(* CoDeSys 2.3.9.41 project: A1.pro *)
(* Libraries: STANDARD.LIB*16.9.21 10:31:38, IECSFC.LIB*16.9.21 10:31:38, SYSLIBTIME.LIB*16.9.21 10:31:38, SYSTASKINFO.LIB*16.9.21 10:31:38, ANALYZATION.LIB*16.9.21 10:31:38, SYSLIBCALLBACK.LIB*16.9.21 10:31:38, Util.lib*16.9.21 10:31:38 *)

(* PLC configuration (modules and I/O channels)
DI_1 AT %IX0.0 [BitInput] Discrete input 1 {ChannellName = Enter name}
DI_2 AT %IX0.1 [BitInput] Discrete input 2 {ChannellName = Enter name}
AT %IB1.0 [ByteInput] 8 discrete inputs {ChannellName = Enter name}
AT %IB1.1 [ByteInput] 8 discrete inputs {ChannellName = Enter name}
DO_1 AT %QX2.0 [BitOutput] Fast discrete output 1 {ChannellName = Enter name}
DO_2 AT %QX2.1 [BitOutput] Fast discrete output 2 {ChannellName = Enter name}
DO_3 AT %QX2.2 [BitOutput] Fast discrete output 3 {ChannellName = Enter name}
DO_4 AT %QX2.3 [BitOutput] Fast discrete output 4 {ChannellName = Enter name}
AT %QB3.0 [ByteOutput] 8 discrete outputs {ChannellName = Enter name}
AT %QB3.1 [ByteOutput] 8 discrete outputs {ChannellName = Enter name}
Special input [ID103] node 4, in %IB4 out %QB4 {ChannellName = Special input}
  AT %IX4.0 [BitInput] Special input {ChannellName = Enter name}
Special output [ID104] node 5, in %IB5 out %QB5 {ChannellName = Special output}
  AT %QX5.0 [BitOutput] Special output {ChannellName = Enter name}
AT %QD6.0 [DWordOutput] Last address {ChannellName = Enter name}
AT %QW6.1 [WordOutput] Last error {ChannellName = Enter name}
RS-485-1 [COM1_USART] node 0, in %IB6.0 out %QB6.0 {ChannellName = RS-485-1; CommunicationSpeed = 115200; Parity = NO PARITY CHECK; BitLength = 8 bits; StopLength = One stop bit; InterfaceType = RS485; FrameOriented = RTU; Timeout = 0; Visibility = No}
AT %QB6.1.0 [ComChannel] Command (0xff - Start) {ChannellName = Enter name}
AlarmA2 AT %QW6.1.0.0 [WordOutput] {ChannellName = Enter name}
qNeedPressure1 AT %QW6.1.1.0 [WordOutput] {ChannellName = Enter name}
qNeedPressure2 AT %QW6.1.2.0 [WordOutput] {ChannellName = Enter name}
qNeedPressure3 AT %QW6.1.3.0 [WordOutput] {ChannellName = Enter name}
iTemp1 AT %QW6.1.4.0 [WordOutput] {ChannellName = Enter name}
iTemp2 AT %QW6.1.5.0 [WordOutput] {ChannellName = Enter name}
iTemp3 AT %QW6.1.6.0 [WordOutput] {ChannellName = Enter name}
iStatusA2 AT %QW6.1.7.0 [WordOutput] {ChannellName = Enter name}
qTempDeltaA2 AT %QW6.1.8.0 [WordOutput] {ChannellName = Enter name}
needAutoAndControlA2 AT %QW6.1.9.0 [WordOutput] {ChannellName = Enter name}
qNeedTempA2 AT %QW6.1.10.0 [WordOutput] {ChannellName = Enter name}
qTime1 AT %QW6.1.11.0 [WordOutput] {ChannellName = Enter name}
qTime2 AT %QW6.1.12.0 [WordOutput] {ChannellName = Enter name}
qTime3 AT %QW6.1.13.0 [WordOutput] {ChannellName = Enter name}
iPressure1 AT %QW6.1.14.0 [WordOutput] {ChannellName = Enter name}
iPressure2 AT %QW6.1.15.0 [WordOutput] {ChannellName = Enter name}
iPressure3 AT %QW6.1.16.0 [WordOutput] {ChannellName = Enter name}
iPressureAll AT %QW6.1.17.0 [WordOutput] {ChannellName = Enter name}
iPressureOil AT %QW6.1.18.0 [WordOutput] {ChannellName = Enter name}
AT %QB6.2.0 [ComChannel] Command (0xff - Start) {ChannellName = Enter name}
AlarmA3 AT %QW6.2.0.0 [WordOutput] {ChannellName = Enter name}
qNeedPressure4 AT %QW6.2.1.0 [WordOutput] {ChannellName = Enter name}
qNeedPressure5 AT %QW6.2.2.0 [WordOutput] {ChannellName = Enter name}
qNeedPressure6 AT %QW6.2.3.0 [WordOutput] {ChannellName = Enter name}
iTemp4 AT %QW6.2.4.0 [WordOutput] {ChannellName = Enter name}
iTemp5 AT %QW6.2.5.0 [WordOutput] {ChannellName = Enter name}
iTemp6 AT %QW6.2.6.0 [WordOutput] {ChannellName = Enter name}
iStatusA3 AT %QW6.2.7.0 [WordOutput] {ChannellName = Enter name}
qTempDeltaA3 AT %QW6.2.8.0 [WordOutput] {ChannellName = Enter name}
needAutoAndControlA3 AT %QW6.2.9.0 [WordOutput] {ChannellName = Enter name}
qNeedTempA3 AT %QW6.2.10.0 [WordOutput] {ChannellName = Enter name}
qTime4 AT %QW6.2.11.0 [WordOutput] {ChannellName = Enter name}
qTime5 AT %QW6.2.12.0 [WordOutput] {ChannellName = Enter name}
qTime6 AT %QW6.2.13.0 [WordOutput] {ChannellName = Enter name}
iPressure4 AT %QW6.2.14.0 [WordOutput] {ChannellName = Enter name}
iPressure5 AT %QW6.2.15.0 [WordOutput] {ChannellName = Enter name}
iPressure6 AT %QW6.2.16.0 [WordOutput] {ChannellName = Enter name}
AT %QD7.0 [DWordOutput] Last address {ChannellName = Enter name}
AT %QW7.1 [WordOutput] Last error {ChannellName = Enter name}
Empty [Empty_module] node 0, in %IB7.0 out %QB7.0 {ChannellName = Empty slot}
AT %QB7.1.0 [ComChannel] Command (0xff - Start) {ChannellName = Enter name}
iNeedTemp AT %QW7.1.0.0 [WordOutput] {ChannellName = Enter name}
qPressure1 AT %QW7.1.1.0 [WordOutput] {ChannellName = Enter name}
qPressure2 AT %QW7.1.2.0 [WordOutput] {ChannellName = Enter name}
qPressure3 AT %QW7.1.3.0 [WordOutput] {ChannellName = Enter name}
qPressure4 AT %QW7.1.4.0 [WordOutput] {ChannellName = Enter name}
qPressure5 AT %QW7.1.5.0 [WordOutput] {ChannellName = Enter name}
qPressure6 AT %QW7.1.6.0 [WordOutput] {ChannellName = Enter name}
iNeedPressure1 AT %QW7.1.7.0 [WordOutput] {ChannellName = Enter name}
iNeedPressure2 AT %QW7.1.8.0 [WordOutput] {ChannellName = Enter name}
iNeedPressure3 AT %QW7.1.9.0 [WordOutput] {ChannellName = Enter name}
iNeedPressure4 AT %QW7.1.10.0 [WordOutput] {ChannellName = Enter name}
iNeedPressure5 AT %QW7.1.11.0 [WordOutput] {ChannellName = Enter name}
iNeedPressure6 AT %QW7.1.12.0 [WordOutput] {ChannellName = Enter name}
qAlarms AT %QW7.1.13.0 [WordOutput] {ChannellName = Enter name}
qTemp1 AT %QW7.1.14.0 [WordOutput] {ChannellName = Enter name}
qTemp2 AT %QW7.1.15.0 [WordOutput] {ChannellName = Enter name}
qTemp3 AT %QW7.1.16.0 [WordOutput] {ChannellName = Enter name}
qTemp4 AT %QW7.1.17.0 [WordOutput] {ChannellName = Enter name}
qTemp5 AT %QW7.1.18.0 [WordOutput] {ChannellName = Enter name}
qTemp6 AT %QW7.1.19.0 [WordOutput] {ChannellName = Enter name}
qPressureAll AT %QW7.1.20.0 [WordOutput] {ChannellName = Enter name}
Register output module [ID2004] node 21, in %IB7.1.21 out %QB7.1.21 {ChannellName = Register; ModbusAddress = 401; Command_write_one_reg = Preset singl register (0x06); Visibility = No}
  qPressureOil AT %QW7.1.21.0 [WordOutput] {ChannellName = Enter name}
Register input module [ID2003] node 22, in %IB7.1.22 out %QB7.1.22 {ChannellName = Register input module; ModbusAddress = 10902; Command_read_regs = Read holding Registers  (0x03); Visibility = No}
  iTempMin AT %QW7.1.22.0 [WordOutput] {ChannellName = Enter name}
Register input module [ID2003] node 23, in %IB7.1.23 out %QB7.1.23 {ChannellName = Register input module; ModbusAddress = 10903; Command_read_regs = Read holding Registers  (0x03); Visibility = No}
  iTempDelta AT %QW7.1.23.0 [WordOutput] {ChannellName = Enter name}
Register input module [ID2003] node 24, in %IB7.1.24 out %QB7.1.24 {ChannellName = Register input module; ModbusAddress = 10904; Command_read_regs = Read holding Registers  (0x03); Visibility = No}
  iPressureOilMax AT %QW7.1.24.0 [WordOutput] {ChannellName = Enter name}
Register input module [ID2003] node 25, in %IB7.1.25 out %QB7.1.25 {ChannellName = Register input module; ModbusAddress = 10905; Command_read_regs = Read holding Registers  (0x03); Visibility = No}
  iPressureAllMax AT %QW7.1.25.0 [WordOutput] {ChannellName = Enter name}
  iTime1 AT %QW7.1.26.0 [WordOutput] {ChannellName = Enter name}
  iTime2 AT %QW7.1.27.0 [WordOutput] {ChannellName = Enter name}
  iTime3 AT %QW7.1.28.0 [WordOutput] {ChannellName = Enter name}
  iTime4 AT %QW7.1.29.0 [WordOutput] {ChannellName = Enter name}
  iTime5 AT %QW7.1.30.0 [WordOutput] {ChannellName = Enter name}
  iTime6 AT %QW7.1.31.0 [WordOutput] {ChannellName = Enter name}
  iAutoStatus AT %QW7.1.32.0 [WordOutput] {ChannellName = Enter name}
*)

(* POU PLC_PRG, CFC *)
PROGRAM PLC_PRG
VAR
	(* DI *)
	AlarmControlIN: BOOL;
	ServiceModeIN: BOOL;
	AlarmStopIN: BOOL;
	AlarmRopeIN: BOOL;
	ControlHydrostationIN: BOOL;
	ControlMotorOilIN: BOOL;
	TENFirstControl: BOOL;
	TENSecondControl: BOOL;
	TENControlTemp: BOOL;
	AlarmVent: BOOL;

	(* DO *)
	AlarmLamp:BOOL;
	AlarmControlLamp:BOOL;
	Hydrostation:BOOL;
	OilMotor:BOOL;
	TEN1:BOOL;
	TEN2:BOOL;


	ControlHydrostation: BOOL;
	ControlMotorOil: BOOL;

	AlarmControl: BOOL;
	ServiceMode: BOOL;
	AlarmStop: BOOL;
	AlarmRope: BOOL;
	Alarms: WORD;
	tenscontroll: TENsControl;
	NotAlarm: BOOL;
	wtb1: WORDToBOOLs;
	wtb2: WORDToBOOLs;
	CloseSec1: BOOL;
	CloseSec2: BOOL;
	CloseSec3: BOOL;
	OpenSec1: BOOL;
	OpenSec2: BOOL;
	OpenSec3: BOOL;
	TempReady1: BOOL;
	TempReady2: BOOL;
	TempReady3: BOOL;
	WorkAcc1: BOOL;
	WorkAcc2: BOOL;
	WorkAcc3: BOOL;
	CloseSec4: BOOL;
	CloseSec5: BOOL;
	CloseSec6: BOOL;
	OpenSec4: BOOL;
	OpenSec5: BOOL;
	OpenSec6: BOOL;
	CloseSec1Auto:BOOL;
	CloseSec2Auto:BOOL;
	CloseSec3Auto:BOOL;
	CloseSec4Auto:BOOL;
	CloseSec5Auto:BOOL;
	CloseSec6Auto:BOOL;
	OpenSec1Auto:BOOL;
	OpenSec2Auto:BOOL;
	OpenSec3Auto:BOOL;
	OpenSec4Auto:BOOL;
	OpenSec5Auto:BOOL;
	OpenSec6Auto:BOOL;


	oilSR: SR;
	tenTON: TON;

	ClosePermission:BOOL;
	OpenPermission:BOOL;
	CloseSRPerm: SR;
	needAutoAndControl: BOOL;
	autoup: UNPACK;
	auto1: BOOL;
	auto2: BOOL;
	auto3: BOOL;
	auto4: BOOL;
	auto5: BOOL;
	auto6: BOOL;
	or101: ORs10FB;
	or102: ORs10FB;
END_VAR
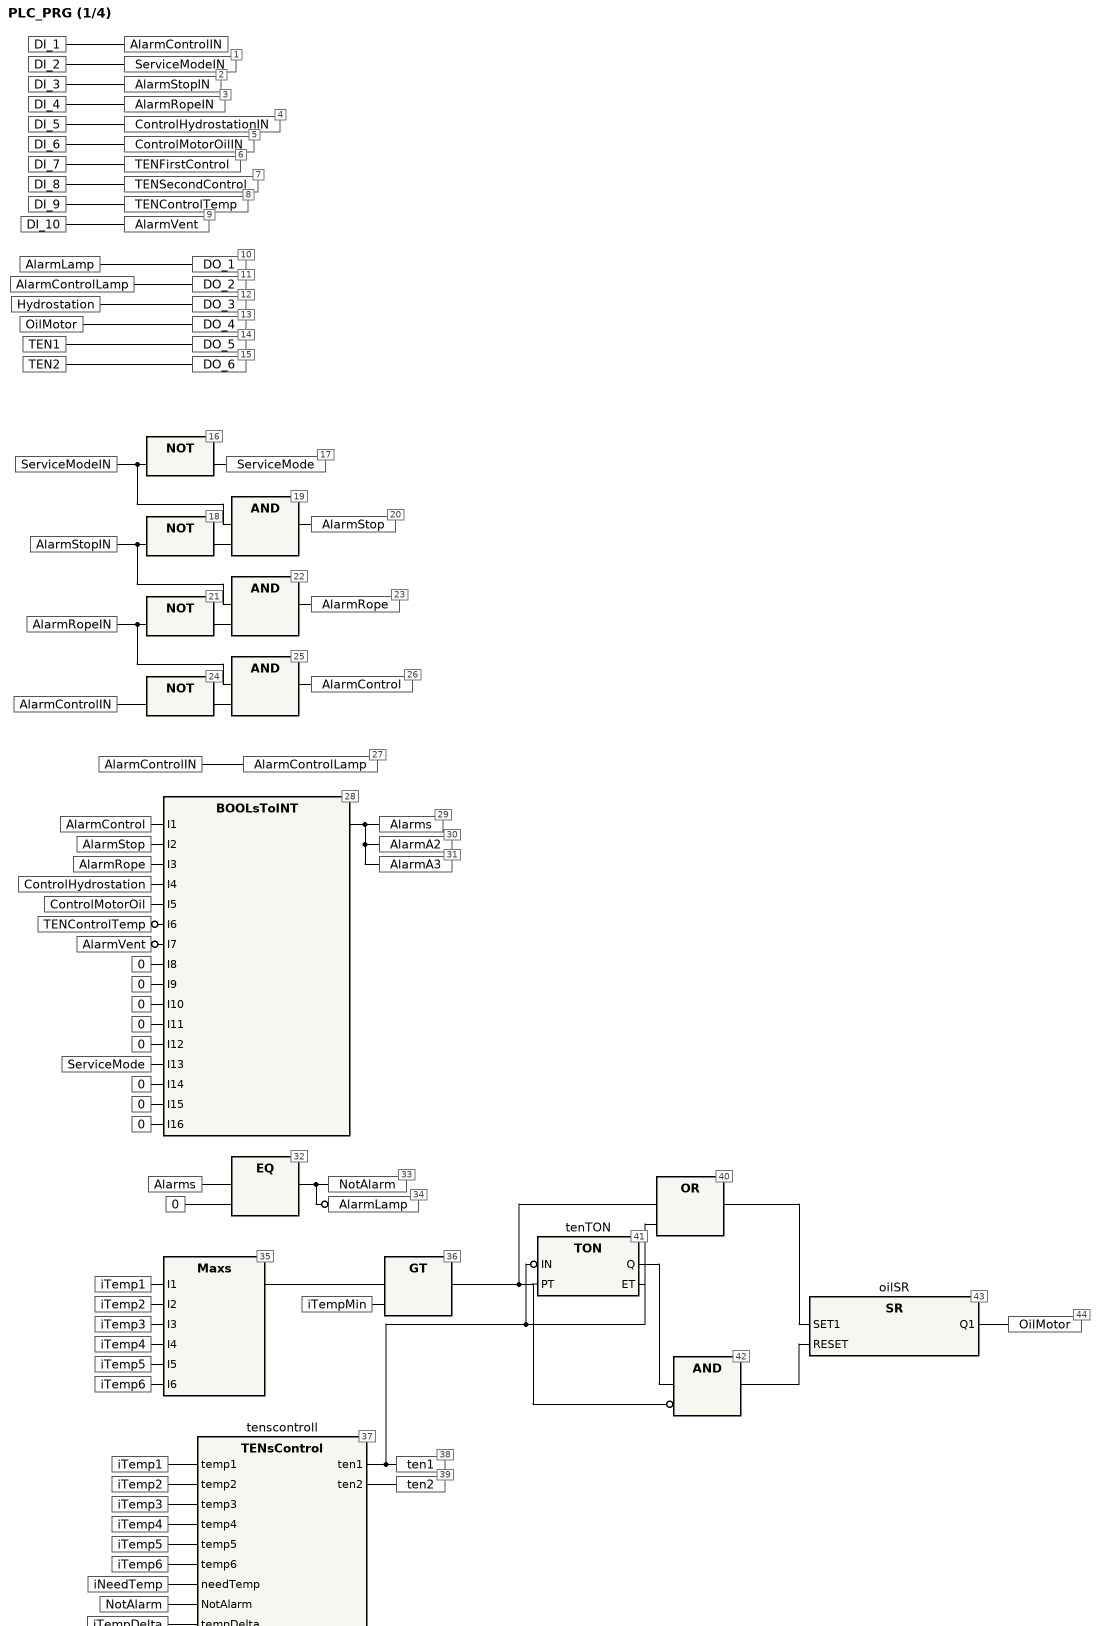
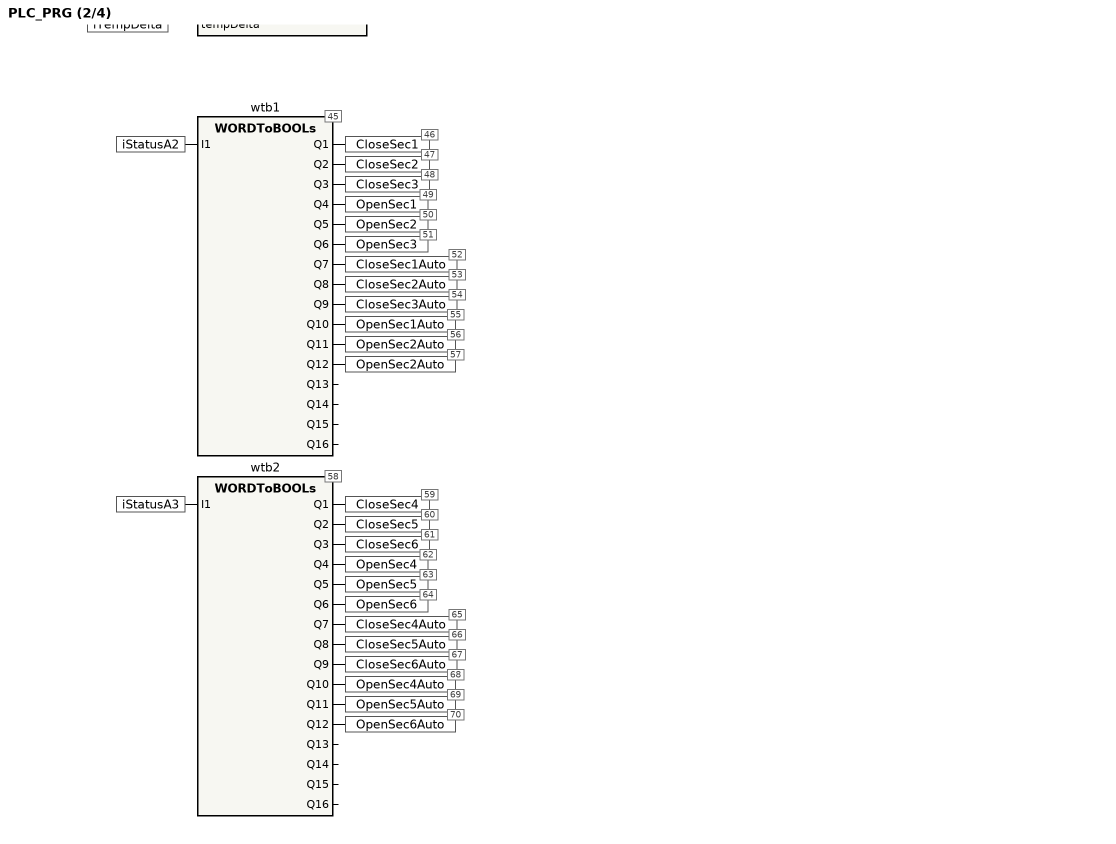
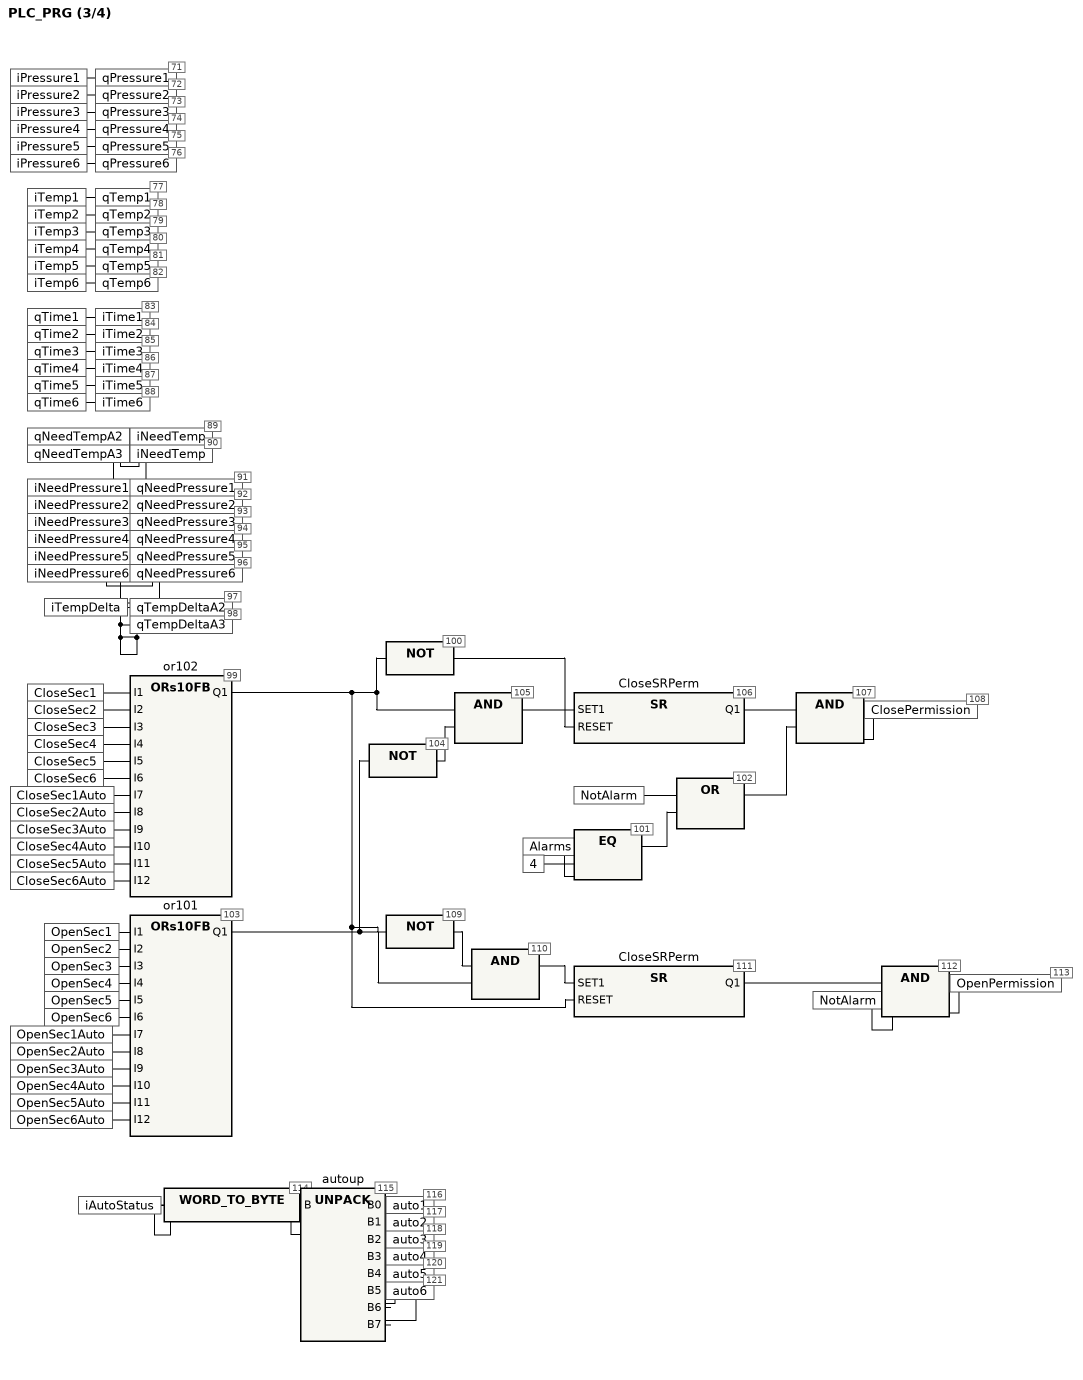
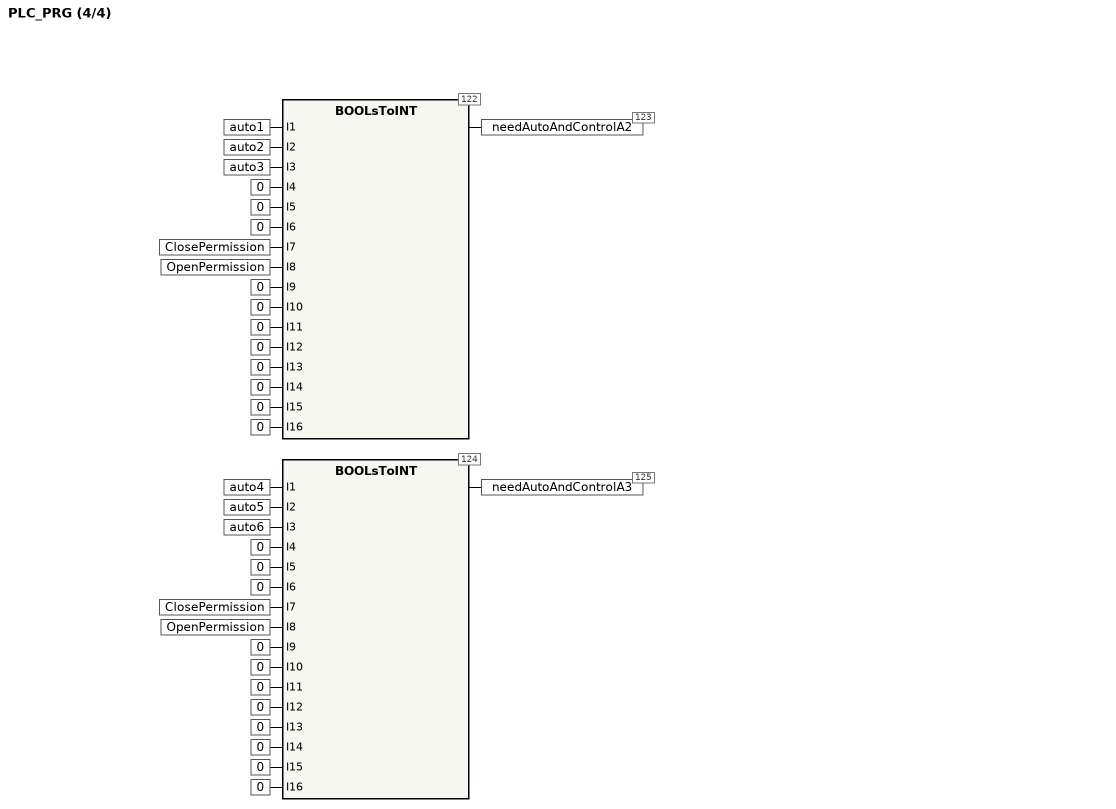
_CFC_ (* Continuous Function Chart, elements in execution order *)
#0 AlarmControlIN <= DI_1
#1 ServiceModeIN <= DI_2
#2 AlarmStopIN <= DI_3
#3 AlarmRopeIN <= DI_4
#4 ControlHydrostationIN <= DI_5
#5 ControlMotorOilIN <= DI_6
#6 TENFirstControl <= DI_7
#7 TENSecondControl <= DI_8
#8 TENControlTemp <= DI_9
#9 AlarmVent <= DI_10
#10 DO_1 <= AlarmLamp
#11 DO_2 <= AlarmControlLamp
#12 DO_3 <= Hydrostation
#13 DO_4 <= OilMotor
#14 DO_5 <= TEN1
#15 DO_6 <= TEN2
#16 NOT(ServiceModeIN)
#17 ServiceMode <= #16
#18 NOT(AlarmStopIN)
#19 AND(ServiceModeIN, #18)
#20 AlarmStop <= #19
#21 NOT(AlarmRopeIN)
#22 AND(AlarmStopIN, #21)
#23 AlarmRope <= #22
#24 NOT(AlarmControlIN)
#25 AND(AlarmRopeIN, #24)
#26 AlarmControl <= #25
#27 AlarmControlLamp <= AlarmControlIN
#28 BOOLsToINT(I1: AlarmControl, I2: AlarmStop, I3: AlarmRope, I4: ControlHydrostation, I5: ControlMotorOil, I6: NOT TENControlTemp, I7: NOT AlarmVent, I8: 0, I9: 0, I10: 0, I11: 0, I12: 0, I13: ServiceMode, I14: 0, I15: 0, I16: 0)
#29 Alarms <= #28
#30 AlarmA2 <= #28
#31 AlarmA3 <= #28
#32 EQ(Alarms, 0)
#33 NotAlarm <= #32
#34 AlarmLamp <= NOT #32
#35 Maxs(I1: iTemp1, I2: iTemp2, I3: iTemp3, I4: iTemp4, I5: iTemp5, I6: iTemp6)
#36 GT(#35, iTempMin)
#37 tenscontroll:TENsControl(temp1: iTemp1, temp2: iTemp2, temp3: iTemp3, temp4: iTemp4, temp5: iTemp5, temp6: iTemp6, needTemp: iNeedTemp, NotAlarm: NotAlarm, tempDelta: iTempDelta)
#38 ten1 <= #37.ten1
#39 ten2 <= #37.ten2
#40 OR(#36, #37.ten1)
#41 tenTON:TON(IN: NOT #37.ten1, PT: -)
#42 AND(#41.Q, NOT #36)
#43 oilSR:SR(SET1: #40, RESET: #42)
#44 OilMotor <= #43.Q1
#45 wtb1:WORDToBOOLs(I1: iStatusA2)
#46 CloseSec1 <= #45.Q1
#47 CloseSec2 <= #45.Q2
#48 CloseSec3 <= #45.Q3
#49 OpenSec1 <= #45.Q4
#50 OpenSec2 <= #45.Q5
#51 OpenSec3 <= #45.Q6
#52 CloseSec1Auto <= #45.Q7
#53 CloseSec2Auto <= #45.Q8
#54 CloseSec3Auto <= #45.Q9
#55 OpenSec1Auto <= #45.Q10
#56 OpenSec2Auto <= #45.Q11
#57 OpenSec2Auto <= #45.Q12
#58 wtb2:WORDToBOOLs(I1: iStatusA3)
#59 CloseSec4 <= #58.Q1
#60 CloseSec5 <= #58.Q2
#61 CloseSec6 <= #58.Q3
#62 OpenSec4 <= #58.Q4
#63 OpenSec5 <= #58.Q5
#64 OpenSec6 <= #58.Q6
#65 CloseSec4Auto <= #58.Q7
#66 CloseSec5Auto <= #58.Q8
#67 CloseSec6Auto <= #58.Q9
#68 OpenSec4Auto <= #58.Q10
#69 OpenSec5Auto <= #58.Q11
#70 OpenSec6Auto <= #58.Q12
#71 qPressure1 <= iPressure1
#72 qPressure2 <= iPressure2
#73 qPressure3 <= iPressure3
#74 qPressure4 <= iPressure4
#75 qPressure5 <= iPressure5
#76 qPressure6 <= iPressure6
#77 qTemp1 <= iTemp1
#78 qTemp2 <= iTemp2
#79 qTemp3 <= iTemp3
#80 qTemp4 <= iTemp4
#81 qTemp5 <= iTemp5
#82 qTemp6 <= iTemp6
#83 iTime1 <= qTime1
#84 iTime2 <= qTime2
#85 iTime3 <= qTime3
#86 iTime4 <= qTime4
#87 iTime5 <= qTime5
#88 iTime6 <= qTime6
#89 iNeedTemp <= qNeedTempA2
#90 iNeedTemp <= qNeedTempA3
#91 qNeedPressure1 <= iNeedPressure1
#92 qNeedPressure2 <= iNeedPressure2
#93 qNeedPressure3 <= iNeedPressure3
#94 qNeedPressure4 <= iNeedPressure4
#95 qNeedPressure5 <= iNeedPressure5
#96 qNeedPressure6 <= iNeedPressure6
#97 qTempDeltaA2 <= iTempDelta
#98 qTempDeltaA3 <= iTempDelta
#99 or102:ORs10FB(I1: CloseSec1, I2: CloseSec2, I3: CloseSec3, I4: CloseSec4, I5: CloseSec5, I6: CloseSec6, I7: CloseSec1Auto, I8: CloseSec2Auto, I9: CloseSec3Auto, I10: CloseSec4Auto, I11: CloseSec5Auto, I12: CloseSec6Auto)
#100 NOT(#99.Q1)
#101 EQ(Alarms, 4)
#102 OR(NotAlarm, #101)
#103 or101:ORs10FB(I1: OpenSec1, I2: OpenSec2, I3: OpenSec3, I4: OpenSec4, I5: OpenSec5, I6: OpenSec6, I7: OpenSec1Auto, I8: OpenSec2Auto, I9: OpenSec3Auto, I10: OpenSec4Auto, I11: OpenSec5Auto, I12: OpenSec6Auto)
#104 NOT(#103.Q1)
#105 AND(#99.Q1, #104)
#106 CloseSRPerm:SR(SET1: #105, RESET: #100)
#107 AND(#106.Q1, #102)
#108 ClosePermission <= #107
#109 NOT(#99.Q1)
#110 AND(#109, #103.Q1)
#111 CloseSRPerm:SR(SET1: #110, RESET: #99.Q1)
#112 AND(#111.Q1, NotAlarm)
#113 OpenPermission <= #112
#114 WORD_TO_BYTE(iAutoStatus)
#115 autoup:UNPACK(B: #114)
#116 auto1 <= #115.B0
#117 auto2 <= #115.B1
#118 auto3 <= #115.B2
#119 auto4 <= #115.B3
#120 auto5 <= #115.B4
#121 auto6 <= #115.B5
#122 BOOLsToINT(I1: auto1, I2: auto2, I3: auto3, I4: 0, I5: 0, I6: 0, I7: ClosePermission, I8: OpenPermission, I9: 0, I10: 0, I11: 0, I12: 0, I13: 0, I14: 0, I15: 0, I16: 0)
#123 needAutoAndControlA2 <= #122
#124 BOOLsToINT(I1: auto4, I2: auto5, I3: auto6, I4: 0, I5: 0, I6: 0, I7: ClosePermission, I8: OpenPermission, I9: 0, I10: 0, I11: 0, I12: 0, I13: 0, I14: 0, I15: 0, I16: 0)
#125 needAutoAndControlA3 <= #124
_END_CFC_
END_PROGRAM

(* POU TENsControl, CFC *)
FUNCTION_BLOCK TENsControl
VAR_INPUT
	temp1:WORD;
	temp2:WORD;
	temp3:WORD;
	temp4:WORD;
	temp5:WORD;
	temp6:WORD;
	needTemp:WORD;
	NotAlarm:BOOL;
	tempDelta:WORD;
END_VAR
VAR_OUTPUT
	ten1:BOOL;
	ten2:BOOL;
END_VAR
VAR
	sss: SR;
END_VAR
VAR (* helpers for the ST form of the networks *)
	_t13 : WORD;
	_t10 : WORD;
	_t12 : BOOL;
	_t17 : BOOL;
	_t18 : BOOL;
	_t14 : WORD;
	_t19 : BOOL;
	_t20 : WORD;
END_VAR
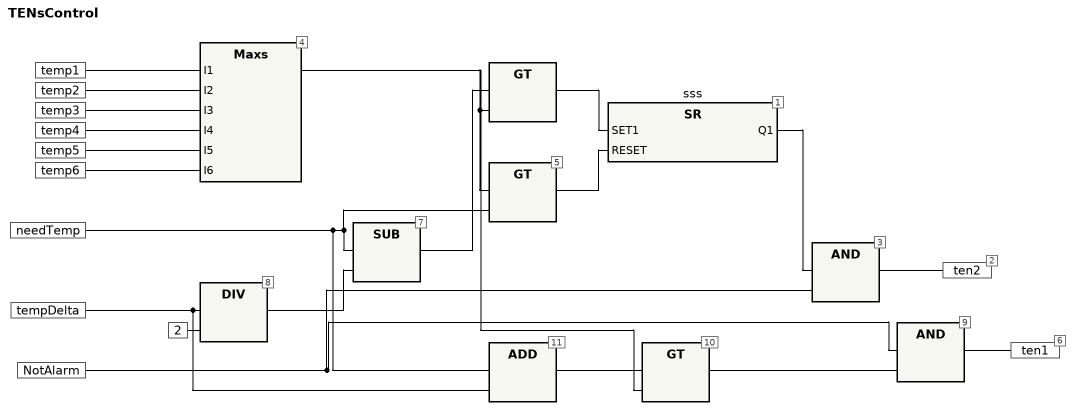
_CFC_ (* Continuous Function Chart, elements in execution order *)
#0 GT(#7, #4)
#1 sss:SR(SET1: #0, RESET: #5)
#2 ten2 <= #3
#3 AND(#1.Q1, NotAlarm)
#4 Maxs(I1: temp1, I2: temp2, I3: temp3, I4: temp4, I5: temp5, I6: temp6)
#5 GT(#4, needTemp)
#6 ten1 <= #9
#7 SUB(needTemp, #8)
#8 DIV(tempDelta, 2)
#9 AND(NotAlarm, #10)
#10 GT(#11, #4)
#11 ADD(needTemp, tempDelta)
_END_CFC_
(* the same logic as Structured Text *)
sss(SET1 := _t13 > _t10, RESET := _t12);
ten2 := _t17;
_t17 := sss.Q1 AND NotAlarm;
_t10 := Maxs(I1 := temp1, I2 := temp2, I3 := temp3, I4 := temp4, I5 := temp5, I6 := temp6);
_t12 := _t10 > needTemp;
ten1 := _t18;
_t13 := needTemp - _t14;
_t14 := tempDelta / 2;
_t18 := NotAlarm AND _t19;
_t19 := _t20 > _t10;
_t20 := needTemp + tempDelta;
END_FUNCTION_BLOCK

(* POU Maxs, CFC *)
FUNCTION Maxs : WORD
VAR_INPUT
	I1:WORD;
	I2:WORD;
	I3:WORD;
	I4:WORD;
	I5:WORD;
	I6:WORD;
END_VAR
VAR
END_VAR
VAR (* helpers for the ST form of the networks *)
	_t17 : WORD;
	_t15 : WORD;
END_VAR
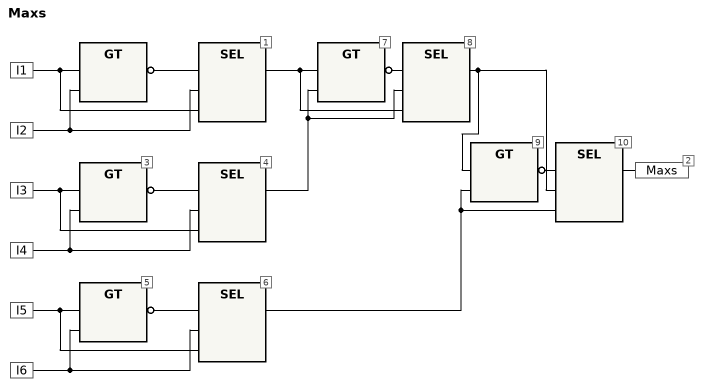
_CFC_ (* Continuous Function Chart, elements in execution order *)
#0 GT(I1, I2)
#1 SEL(NOT #0, I1, I2)
#2 Maxs <= #10
#3 GT(I3, I4)
#4 SEL(NOT #3, I3, I4)
#5 GT(I5, I6)
#6 SEL(NOT #5, I5, I6)
#7 GT(#1, #4)
#8 SEL(NOT #7, #1, #4)
#9 GT(#8, #6)
#10 SEL(NOT #9, #8, #6)
_END_CFC_
(* the same logic as Structured Text *)
Maxs := _t17;
_t15 := SEL(NOT (SEL(NOT (I1 > I2), I1, I2) > SEL(NOT (I3 > I4), I3, I4)), SEL(NOT (I1 > I2), I1, I2), SEL(NOT (I3 > I4), I3, I4));
_t17 := SEL(NOT (_t15 > SEL(NOT (I5 > I6), I5, I6)), _t15, SEL(NOT (I5 > I6), I5, I6));
END_FUNCTION

(* POU WORDToBOOLs, CFC *)
FUNCTION_BLOCK WORDToBOOLs
VAR_INPUT
	I1:WORD;
END_VAR
VAR_OUTPUT
	Q1:BOOL;
	Q2:BOOL;
	Q3:BOOL;
	Q4:BOOL;
	Q5:BOOL;
	Q6:BOOL;
	Q7:BOOL;
	Q8:BOOL;
	Q9:BOOL;
	Q10:BOOL;
	Q11:BOOL;
	Q12:BOOL;
	Q13:BOOL;
	Q14:BOOL;
	Q15:BOOL;
	Q16:BOOL;
END_VAR
VAR
	unp1: UNPACK;
	unp2: UNPACK;
END_VAR
VAR (* helpers for the ST form of the networks *)
	_t28 : BYTE;
	_t31 : BYTE;
END_VAR
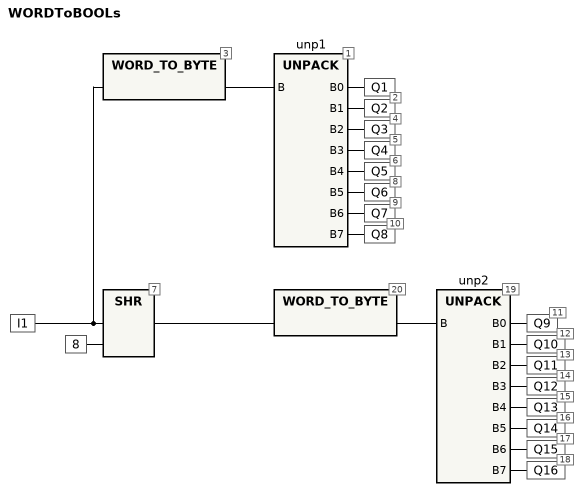
_CFC_ (* Continuous Function Chart, elements in execution order *)
#0 Q1 <= #1.B0
#1 unp1:UNPACK(B: #3)
#2 Q2 <= #1.B1
#3 WORD_TO_BYTE(I1)
#4 Q3 <= #1.B2
#5 Q4 <= #1.B3
#6 Q5 <= #1.B4
#7 SHR(I1, 8)
#8 Q6 <= #1.B5
#9 Q7 <= #1.B6
#10 Q8 <= #1.B7
#11 Q9 <= #19.B0
#12 Q10 <= #19.B1
#13 Q11 <= #19.B2
#14 Q12 <= #19.B3
#15 Q13 <= #19.B4
#16 Q14 <= #19.B5
#17 Q15 <= #19.B6
#18 Q16 <= #19.B7
#19 unp2:UNPACK(B: #20)
#20 WORD_TO_BYTE(#7)
_END_CFC_
(* the same logic as Structured Text *)
Q1 := unp1.B0;
unp1(B := _t28);
Q2 := unp1.B1;
_t28 := WORD_TO_BYTE(I1);
Q3 := unp1.B2;
Q4 := unp1.B3;
Q5 := unp1.B4;
Q6 := unp1.B5;
Q7 := unp1.B6;
Q8 := unp1.B7;
Q9 := unp2.B0;
Q10 := unp2.B1;
Q11 := unp2.B2;
Q12 := unp2.B3;
Q13 := unp2.B4;
Q14 := unp2.B5;
Q15 := unp2.B6;
Q16 := unp2.B7;
unp2(B := _t31);
_t31 := WORD_TO_BYTE(SHR(I1, 8));
END_FUNCTION_BLOCK

(* POU ORs10FB, ST *)
FUNCTION_BLOCK ORs10FB
VAR_INPUT
	I1: BOOL;
	I2: BOOL;
	I3: BOOL;
	I4: BOOL;
	I5: BOOL;
	I6: BOOL;
	I7: BOOL;
	I8: BOOL;
	I9: BOOL;
	I10 :BOOL;
	I11 :BOOL;
	I12: BOOL;
END_VAR
VAR_OUTPUT
	Q1: BOOL;
END_VAR
VAR
END_VAR
Q1:=(I1 OR I2) OR (I3 OR I4) OR (I5 OR I6) OR (I7 OR I8) OR (I9 OR I10) OR (I11 OR I12);
END_FUNCTION_BLOCK

(* POU BOOLsToINT, CFC *)
FUNCTION BOOLsToINT : WORD
VAR_INPUT
	I1:BOOL;
	I2:BOOL;
	I3:BOOL;
	I4:BOOL;
	I5:BOOL;
	I6:BOOL;
	I7:BOOL;
	I8:BOOL;
	I9:BOOL;
	I10:BOOL;
	I11:BOOL;
	I12:BOOL;
	I13:BOOL;
	I14:BOOL;
	I15:BOOL;
	I16:BOOL;
END_VAR
VAR
END_VAR
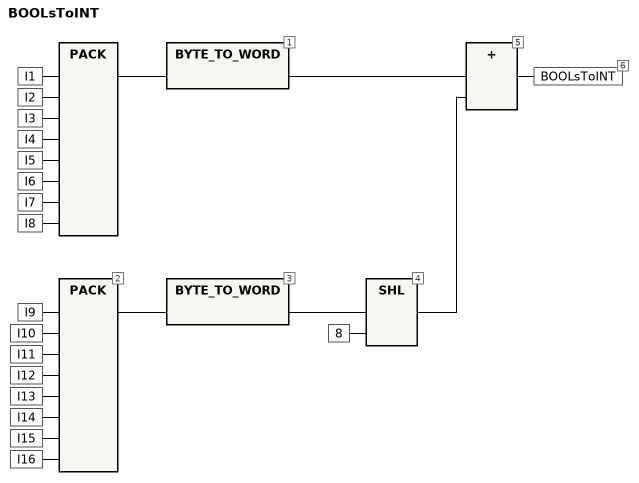
_CFC_ (* Continuous Function Chart, elements in execution order *)
#0 PACK(I1, I2, I3, I4, I5, I6, I7, I8)
#1 BYTE_TO_WORD(#0)
#2 PACK(I9, I10, I11, I12, I13, I14, I15, I16)
#3 BYTE_TO_WORD(#2)
#4 SHL(#3, 8)
#5 +(#1, #4)
#6 BOOLsToINT <= #5
_END_CFC_
END_FUNCTION

(* POU ORs10ST, ST *)
FUNCTION ORs10ST : BOOL
VAR_INPUT
	I1:BOOL;
	I2:BOOL;
	I3:BOOL;
	I4:BOOL;
	I5:BOOL;
	I6:BOOL;
	I7:BOOL;
	I8:BOOL;
	I9:BOOL;
	I10:BOOL;
	I11:BOOL;
	I12:BOOL;
END_VAR
VAR
END_VAR
ORs10ST:=I1 OR I2 OR I3 OR I4 OR I5 OR I6 OR I7 OR I8 OR I9 OR I10 OR I11 OR I12;
END_FUNCTION
